FUNCTION_BLOCK BatterySensor (* Sensor for receiving data from the BatterySensor plugin controller in Polysun *)
  (* Standard: 61499-2 *)
  (* Version 1.0, 2017-07-21, Marc Jakobi, HTW Berlin *)
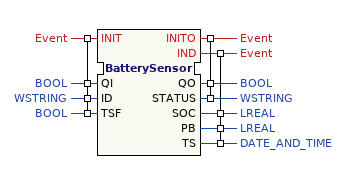
  EVENT_INPUT
    INIT WITH QI, ID, TSF; (* Initialization Request *)
  END_EVENT
  EVENT_OUTPUT
    INITO WITH QO, STATUS; (* Initialization Confirm *)
    IND WITH SOC, PB, TS; (* Execution Confirmation *)
  END_EVENT
  VAR_INPUT
    QI : BOOL; (* Input event qualifier *)
    ID : WSTRING; (* Connection identifier *)
    TSF : BOOL; (* Flag for whether to receive time stamp or not *)
  END_VAR
  VAR_OUTPUT
    QO : BOOL; (* Output event qualifier *)
    STATUS : WSTRING; (* Service status *)
    SOC : LREAL; (* State of charge [0,..,1] *)
    PB : LREAL; (* Battery transfer in W *)
    TS : DATE_AND_TIME; (* Time stamp (optional) *)
  END_VAR
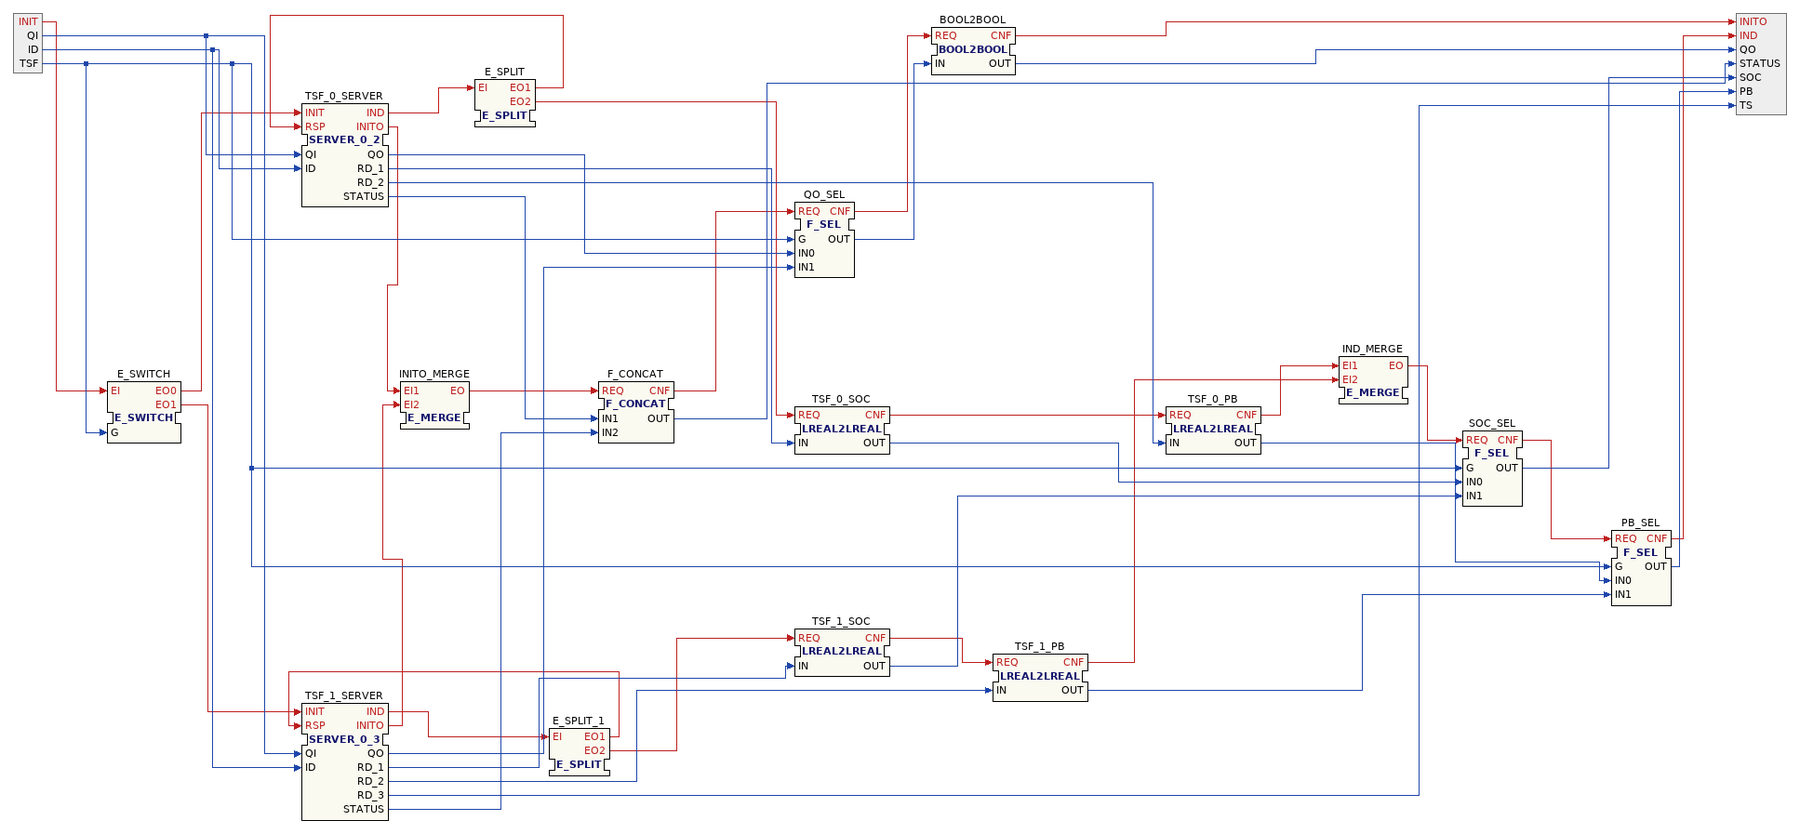
  FBS
    TSF_1_SERVER : SERVER_0_3;
    TSF_0_SERVER : SERVER_0_2;
    E_SWITCH : E_SWITCH;
    E_SPLIT : E_SPLIT;
    E_SPLIT_1 : E_SPLIT;
    INITO_MERGE : E_MERGE;
    IND_MERGE : E_MERGE;
    QO_SEL : F_SEL;
    SOC_SEL : F_SEL;
    TSF_0_SOC : LREAL2LREAL;
    TSF_1_SOC : LREAL2LREAL;
    TSF_0_PB : LREAL2LREAL;
    TSF_1_PB : LREAL2LREAL;
    PB_SEL : F_SEL;
    BOOL2BOOL : BOOL2BOOL;
    F_CONCAT : F_CONCAT;
  END_FBS
  EVENT_CONNECTIONS
    INIT TO E_SWITCH.EI;
    E_SWITCH.EO0 TO TSF_0_SERVER.INIT;
    E_SWITCH.EO1 TO TSF_1_SERVER.INIT;
    E_SPLIT.EO1 TO TSF_0_SERVER.RSP;
    TSF_1_SERVER.IND TO E_SPLIT_1.EI;
    E_SPLIT_1.EO1 TO TSF_1_SERVER.RSP;
    E_SPLIT.EO2 TO TSF_0_SOC.REQ;
    E_SPLIT_1.EO2 TO TSF_1_SOC.REQ;
    TSF_0_SOC.CNF TO TSF_0_PB.REQ;
    TSF_1_SOC.CNF TO TSF_1_PB.REQ;
    TSF_0_PB.CNF TO IND_MERGE.EI1;
    TSF_1_PB.CNF TO IND_MERGE.EI2;
    IND_MERGE.EO TO SOC_SEL.REQ;
    SOC_SEL.CNF TO PB_SEL.REQ;
    PB_SEL.CNF TO IND;
    QO_SEL.CNF TO BOOL2BOOL.REQ;
    TSF_0_SERVER.IND TO E_SPLIT.EI;
    TSF_0_SERVER.INITO TO INITO_MERGE.EI1;
    TSF_1_SERVER.INITO TO INITO_MERGE.EI2;
    INITO_MERGE.EO TO F_CONCAT.REQ;
    F_CONCAT.CNF TO QO_SEL.REQ;
    BOOL2BOOL.CNF TO INITO;
  END_CONNECTIONS
  DATA_CONNECTIONS
    QI TO TSF_1_SERVER.QI;
    QI TO TSF_0_SERVER.QI;
    ID TO TSF_1_SERVER.ID;
    ID TO TSF_0_SERVER.ID;
    TSF TO E_SWITCH.G;
    TSF TO QO_SEL.G;
    TSF_0_SERVER.QO TO QO_SEL.IN0;
    TSF_1_SERVER.QO TO QO_SEL.IN1;
    TSF TO SOC_SEL.G;
    TSF_0_SERVER.RD_1 TO TSF_0_SOC.IN;
    TSF_1_SERVER.RD_1 TO TSF_1_SOC.IN;
    TSF_0_SOC.OUT TO SOC_SEL.IN0;
    TSF_1_SOC.OUT TO SOC_SEL.IN1;
    TSF_0_SERVER.RD_2 TO TSF_0_PB.IN;
    TSF_1_SERVER.RD_2 TO TSF_1_PB.IN;
    TSF_1_SERVER.RD_3 TO TS;
    TSF TO PB_SEL.G;
    TSF_0_PB.OUT TO PB_SEL.IN0;
    TSF_1_PB.OUT TO PB_SEL.IN1;
    SOC_SEL.OUT TO SOC;
    PB_SEL.OUT TO PB;
    QO_SEL.OUT TO BOOL2BOOL.IN;
    BOOL2BOOL.OUT TO QO;
    TSF_0_SERVER.STATUS TO F_CONCAT.IN1;
    TSF_1_SERVER.STATUS TO F_CONCAT.IN2;
    F_CONCAT.OUT TO STATUS;
  END_CONNECTIONS
END_FUNCTION_BLOCK
